# EPICS autosave request: calc/calcApp/Db/calcout_settings.req
# FILE... calcout_settings.req
# USAGE.. calcout Record fields autosave'd.
$(P).A
$(P).B
$(P).C
$(P).D
$(P).E
$(P).F
$(P).G
$(P).H
$(P).I
$(P).J
$(P).K
$(P).L
$(P).INPA
$(P).INPB
$(P).INPC
$(P).INPD
$(P).INPE
$(P).INPF
$(P).INPG
$(P).INPH
$(P).INPI
$(P).INPJ
$(P).INPK
$(P).INPL
$(P).CALC$
$(P).OCAL$
$(P).SCAN
$(P).PREC
$(P).ODLY
$(P).OEVT
$(P).OOPT
$(P).DOPT
$(P).IVOA
$(P).IVOV
$(P).OUT
$(P).FLNK
$(P).DESC
$(P).EVNT
$(P).EGU
